RESOURCE_TYPE VIEW_PANEL (* Container for View elements *)
  (* Standard: 61499-1; Classification: HMI *)
  (* Version 0.0, 2002-04-04, JHC, Rockwell Automation, Derived from PANEL_RESOURCE. *)
  (* Compiler header: package fb.rt.hmi; import java.awt.*; *)
  (* Compiler Java IBM VisualAge 3.0 *)
  VAR_INPUT
    TRACE : BOOL; (* True=trace enabled,default is false *)
    BKGD : COLOR := COLOR#white; (* Background color *)
    DIA : UINT := 25; (* Characteristic dimension,Overrides component DIAs *)
    SIZE : ARRAY [0..1] OF UINT := [2,2]; (* [width,height]in DIA units *)
    VERTICAL : BOOL; (* 1=Column-first,0=Row-first *)
  END_VAR
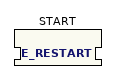
  FBS
    START : E_RESTART;
  END_FBS
END_RESOURCE_TYPE
